TYPE ST_SpraybarErrors :
STRUCT
	NCAxisError						: ST_NcAxis_Errors;
	PositionAtFrontError			: BOOL;	//Zeestra 20190222
	PositionAtBackError				: BOOL;	//Zeestra 20190222
END_STRUCT
END_TYPE

(* stored: Version 1.1.0.1, ProductVersion 3.1.4020.12
   DUT ST_SpraybarErrors: Id {7714b2e4-7067-45cb-8cc2-6c847501c321} *)
